SUBAPPLICATION Uebung_006f_SR (* Exercise for FB_SR_T_FF (Set-Dominant Toggle Flip-Flop) *)
  (* Standard: 61499-2; Description: Copyright (c) 2026 Meisterschulen am Ostbahnhof *)
  (* Version 1.0, 2026-05-07, Gemini CLI, Meisterschulen am Ostbahnhof *)
  PACKAGE Uebungen;
  IMPORT logiBUS::io::DI::logiBUS_DI::Input_I1;
  IMPORT logiBUS::io::DI::logiBUS_DI::Input_I2;
  IMPORT logiBUS::io::DI::logiBUS_DI::Input_I3;
  IMPORT logiBUS::io::DQ::logiBUS_DO::Output_Q1;
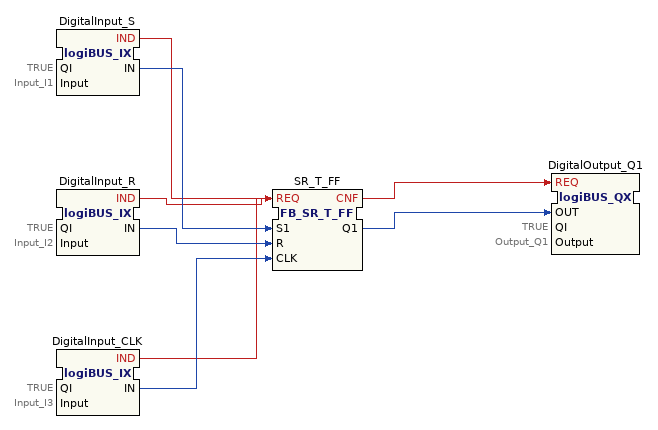
  FBS
    DigitalInput_S : logiBUS::io::DI::logiBUS_IX(QI := TRUE, Input := Input_I1);
    DigitalInput_R : logiBUS::io::DI::logiBUS_IX(QI := TRUE, Input := Input_I2);
    DigitalInput_CLK : logiBUS::io::DI::logiBUS_IX(QI := TRUE, Input := Input_I3);
    SR_T_FF : logiBUS::bistableElements::FB_SR_T_FF;
    DigitalOutput_Q1 : logiBUS::io::DQ::logiBUS_QX(QI := TRUE, Output := Output_Q1);
  END_FBS
  EVENT_CONNECTIONS
    DigitalInput_S.IND TO SR_T_FF.REQ;
    DigitalInput_R.IND TO SR_T_FF.REQ;
    DigitalInput_CLK.IND TO SR_T_FF.REQ;
    SR_T_FF.CNF TO DigitalOutput_Q1.REQ;
  END_CONNECTIONS
  DATA_CONNECTIONS
    DigitalInput_S.IN TO SR_T_FF.S1;
    DigitalInput_R.IN TO SR_T_FF.R;
    DigitalInput_CLK.IN TO SR_T_FF.CLK;
    SR_T_FF.Q1 TO DigitalOutput_Q1.OUT;
  END_CONNECTIONS
END_SUBAPPLICATION
